// TIA Portal V20 export
TYPE "LKinCtrl_typeJogConfiguration"
// stored: Access Published
   STRUCT
      accelerationTime { ExternalAccessible := 'False'; ExternalVisible := 'False'; ExternalWritable := 'False'; S7_SetPoint := 'True'} : LReal;   // Maximum acceleration and deceleration time. while jogging in WCS, OCS1-3, TCS, Axes, MCS and Approach point linear.
      maxVelocityManual { ExternalAccessible := 'False'; ExternalVisible := 'False'; ExternalWritable := 'False'; S7_SetPoint := 'True'} : LReal;
      maxVelocityTestRun { ExternalAccessible := 'False'; ExternalVisible := 'False'; ExternalWritable := 'False'; S7_SetPoint := 'True'} : LReal;
      presetIncrementCoarse { ExternalAccessible := 'False'; ExternalVisible := 'False'; ExternalWritable := 'False'; S7_SetPoint := 'True'} : LReal;
      presetIncrementFine { ExternalAccessible := 'False'; ExternalVisible := 'False'; ExternalWritable := 'False'; S7_SetPoint := 'True'} : LReal;
      presetIncrementPrecise { ExternalAccessible := 'False'; ExternalVisible := 'False'; ExternalWritable := 'False'; S7_SetPoint := 'True'} : LReal;
   END_STRUCT;
END_TYPE
